(* IEC 61131-3 sources: eCockpitGit/test_project/src/%F%00 Library/%F%Common Functions/%F%Buffer, 3 files *)

(* ---- %POU%FU_ClearData.st ---- *)
FUNCTION FU_ClearData : BOOL
VAR_INPUT
	data		:ANY;
END_VAR

(*%!%__DELIMITER__%!%*)
WHILE data.diSize > 0 DO
	data.pValue^		:=		0;
	data.pValue			:=		data.pValue + 1;
	data.diSize			:=		data.diSize - 1;
END_WHILE

(* ---- %POU%FB_FIFOArray.st ---- *)
//Thread safe FIFO array buffer manager
//It can be instanciated simply like below
//	fifo				:FB_FIFOQueue := (S_bufferSize:=SIZEOF(fifoQueue) / SIZEOF(fifoQueue[1]));
//	fifoQueue			:ARRAY[0..10] OF DWORD;
// |**Version**|**Author**| **Date** |**Changes**
// | 1         | NSN      | 15-02-22 | Creation
FUNCTION_BLOCK FB_FIFOArray
VAR_INPUT
	S_startIndex	:DWORD;					//Index of first element in array, only positive indexes are supported
	S_bufferSize	:DWORD;					//Maximum amount of elements in buffer array
END_VAR
VAR
	S_amount		:DWORD;					//How many elements are in the queue
	S_input			:DWORD := 4294967295;	//Last input/push index
	S_output		:DWORD := 4294967295;	//Last output/unshift index
	S_block			:DWORD;					//Block for threadsafeness
	S_blockInput	:DWORD;					//Block for threadsafeness
	S_blockOutput	:DWORD;					//Block for threadsafeness
END_VAR
(*%!%__DELIMITER__%!%*)

(* ---- %POU%FB_FIFOQueue.st ---- *)
//Thread safe FIFO buffer manager
//It can be instanciated simply like below
//	fifo				:FB_FIFOQueue := (S_buffer:=ADR(fifoQueue),S_bufferSize:=SIZEOF(fifoQueue) / SIZEOF(fifoQueue[1]),S_elementSize:=SIZEOF(fifoQueue[1]));
//	fifoQueue			:ARRAY[1..10] OF DWORD;
// |**Version**|**Author**| **Date** |**Changes**
// | 1         | NSN      | 15-02-22 | Creation
FUNCTION_BLOCK FB_FIFOQueue
VAR_INPUT
	S_buffer		:POINTER TO BYTE;		//Reference to buffer
	S_bufferSize	:DWORD;					//Maximum amount of elements in buffer array
	S_elementSize	:DWORD;					//Size of element
END_VAR
VAR
	S_amount		:DWORD;					//How many elements are in the queue
	S_input			:DWORD := 4294967295;	//Last input/push index/offset
	S_output		:DWORD := 4294967295;	//Last output/unshift index/offset
	S_block			:DWORD;					//Block for threadsafeness
	S_blockInput	:DWORD;					//Block for threadsafeness
	S_blockOutput	:DWORD;					//Block for threadsafeness
END_VAR
(*%!%__DELIMITER__%!%*)
